Fanuc KAREL source: compact_preamble.KL

PROGRAM KT00193
%NOLOCKGROUP
VAR
B1:BOOLEAN;B2:BOOLEAN;OUT:BOOLEAN
BEGIN
B1=TRUE
B2=FALSE
B1=TRUE
B2=FALSE
OUT=(B1 AND B2)
END KT00193
